INTERFACE ITF_IOLamp EXTENDS ITF_BaseComponent

(*			
	EVERDE sp. z o.o.
	Rafał Osajda		05.02.2025		TC 4026.13		wer. 0.0.0.1
	Sterowanie swieceniem lampki - włącz/wyłącz
*)
METHOD Control
VAR_INPUT
	bIN						: BOOL;
END_VAR
END_METHOD

(*			
	EVERDE sp. z o.o.
	Rafał Osajda		05.02.2025		TC 4026.13		wer. 0.0.0.1
	Zwraca czy lampka wlaczona
*)
METHOD IsActive : BOOL
END_METHOD

(*			
	EVERDE sp. z o.o.
	Rafał Osajda		05.02.2025		TC 4026.13		wer. 0.0.0.1
	Wylacza lampke
*)
METHOD SetOff
END_METHOD

(*			
	EVERDE sp. z o.o.
	Rafał Osajda		05.02.2025		TC 4026.13		wer. 0.0.0.1
	Wlacza lampke
*)
METHOD SetOn
END_METHOD

END_INTERFACE

(* stored: Version 1.1.0.1
   Itf ITF_IOLamp: Id {f4ae548f-51c7-4567-ab3b-19d520794750}
   Method Control: Id {17fe7be7-aa53-4918-8006-7c621311eb32}
   Method IsActive: Id {bfce1990-4236-49dc-a250-279de524c5da}
   Method SetOff: Id {c6a94966-2135-4e57-84da-cf7100566012}
   Method SetOn: Id {41fac941-ca6b-40a9-a7f8-2a363b15b32a} *)
